TYPE Mat67 : ARRAY[1..6, 1..7] OF LREAL; END_TYPE

(* stored: Version 1.1.0.1, ProductVersion 3.1.4024.12
   DUT Mat67: Id {f8e72d6d-377a-4414-aa2e-dd45756b42be} *)
